(* IEC 61131-3 sources: ST/projects, 7 files *)

(* ---- blink.st ---- *)
PROGRAM PLC_PRG
VAR
start :BOOL; //type declaration
stop  :BOOL;
motor :BOOL;
END_VAR

//loop block
IF start=TRUE THEN  //standard if structure
	motor:=TRUE;
	ELSE
	motor:=FALSE;
END_IF

(* ---- case-of.st ---- *)
PROGRAM PLC_PRG
VAR
	number : INT := 0;
	lamp1  : BOOL;
	lamp2  : BOOL;
	lamp3  : BOOL;
END_VAR

CASE number OF
	1 : lamp1 := TRUE;
	 	lamp2 := FALSE;
		lamp3 := FALSE;

	2 : lamp1 := FALSE;
	 	lamp2 := TRUE;
		lamp3 := FALSE;

	3 : lamp1 := FALSE;
	 	lamp2 := FALSE;
		lamp3 := TRUE;

	ELSE
		lamp1 := FALSE;
	 	lamp2 := FALSE;
		lamp3 := FALSE;
END_CASE

END_PROGRAM

(* ---- count-up-project.st ---- *)
PROGRAM PLC_PRG

VAR
	sensor        :BOOL:=FALSE;
	reset         :BOOL:=FALSE;
	motor         :BOOL;
	counter1      :CTU;
	counterValue  :WORD;
END_VAR

counter1(CU:=sensor, RESET:=reset, PV:=4);
motor := counter1.Q;
counterValue := counter1.CV;

END_PROGRAM

(* ---- for-loop.st ---- *)
PROGRAM PLC_PRG
VAR
	list:ARRAY[0..4] OF REAL:=[10, 20, 30, 40, 50];
	average  : REAL:=0;
	i        : INT :=0;
END_VAR

average:=0;
FOR i:=0 TO 4 DO
	average := average + list[i];
END_FOR

average := average / 5;
END_PROGRAM

(* ---- on-delay-timer.st ---- *)
PROGRAM PLC_PRG

VAR
	timer1       :TON;
	start        :BOOL;
	motor        :BOOL;
	elapsed_time :TIME;
END_VAR

timer1(IN:=start, PT:=T#10S);
elapsed_time:= timer1.ET;
motor:=timer1.Q;

IF start=TRUE THEN
	timer1.IN:=TRUE;
ELSE
	timer1.IN:=FALSE;
END_IF

END_PROGRAM

(* ---- sealing.st ---- *)
PROGRAM PLC_PRG
VAR
	over_current :BOOL;
	stop         :BOOL;
	start        :BOOL;
	motor        :BOOL;
END_VAR

motor:= (over_current AND stop) AND (start OR motor);
END_PROGRAM

(* ---- setReset.st ---- *)
PROGRAM PLC_PRG
VAR
	motor :BOOL;
	start :BOOL;
	stop  :BOOL;
END_VAR

motor S=start;
motor R=stop;

END_PROGRAM
